INTERFACE ITF_Valve2

METHOD Abort : BOOL
VAR_INPUT
END_VAR
END_METHOD

PROPERTY Auto : BOOL
GET
END_GET
SET
END_SET
END_PROPERTY

METHOD Clear : BOOL
VAR_INPUT
END_VAR
END_METHOD

METHOD Close : BOOL
VAR_INPUT
END_VAR
END_METHOD

PROPERTY Error_State  : E_Motor_Error_State
GET
END_GET
END_PROPERTY

PROPERTY Manueel : BOOL
GET
END_GET
SET
END_SET
END_PROPERTY

METHOD Open : BOOL
VAR_INPUT
END_VAR
END_METHOD

METHOD Reset : BOOL
VAR_INPUT
END_VAR
END_METHOD

METHOD Start : BOOL
VAR_INPUT
END_VAR
END_METHOD

PROPERTY State : E_Motor_State
GET
END_GET
END_PROPERTY

METHOD Stop : BOOL
VAR_INPUT
END_VAR
END_METHOD

PROPERTY Tag : STRING
GET
END_GET
END_PROPERTY

END_INTERFACE

(* stored: Version 1.1.0.1, ProductVersion 3.1.4024.12
   Itf ITF_Valve2: Id {44a150d9-ab3f-4358-9804-e0358d103d22}
   Folder Methods: Id {f9cc074a-35ca-4c1f-bf78-aae5d38774fd}
   Folder Properties: Id {f5102dc7-4430-454c-ab58-31e404fa52f2}
   Method Abort: Id {c8fb51d2-c00f-4bf9-b401-2beaf77854fb}
   Property Auto: Id {75c8b575-8f2f-47b4-a957-fc4532666a55}
   Get Get: Id {9f0d31a8-f54e-46be-b783-83d8261f9fcd}
   Set Set: Id {a839cc47-5e29-48bc-b415-c791091eeb7f}
   Method Clear: Id {ddbe7526-07fc-4b10-9385-6013d18aca2b}
   Method Close: Id {14fc7614-d1b6-4aa2-9b4f-7973b30937fe}
   Property Error_State: Id {cd041877-81eb-49bc-a6a3-42222ca31f93}
   Get Get: Id {3c21c68b-4ebc-4c76-93e8-a0b3d78e1a8b}
   Property Manueel: Id {65193eac-4d20-4951-bf46-b829b02da879}
   Get Get: Id {96b50a32-d098-4ede-b777-837ac9494e97}
   Set Set: Id {52b90226-38d7-436e-81ea-c5cfbf2ccae2}
   Method Open: Id {083aea2b-c2b9-45bd-b8fd-6c3a7c65dd42}
   Method Reset: Id {ad596ef7-ffce-49af-a5c5-bfa86c5452e2}
   Method Start: Id {58eebfbe-0f04-4cbe-b793-72e8966ecbad}
   Property State: Id {a2623f99-3364-44c9-b4b8-82b45bd7dfbb}
   Get Get: Id {36439565-1469-4ad7-af72-ca4db3d78844}
   Method Stop: Id {0e4c4af0-ddda-4d58-8442-239e443fbb82}
   Property Tag: Id {5bb1604b-e4f7-460a-904c-d2751008ab91}
   Get Get: Id {13187376-1d21-4f77-8542-b2383e37c132} *)
